PROGRAM EM03_PlacingArea_2
VAR
//----Motor-----
	// Box Placing Roller Conveyor 2	
	FB_BoxPlacingRollerConv_2			: MotorManagement;
	stBoxPlacingRollerConv_2			: stMotor;
	BoxPlacingRollerConv_2_ErrorID		: UINT;
	BoxPlacingRollerConv_2_Error		: BOOL;
	bFL_BoxPlacingRollerConv_2_Forward	: BOOL;
	bFL_BoxPlacingRollerConv_2_Reverse	: BOOL;
END_VAR

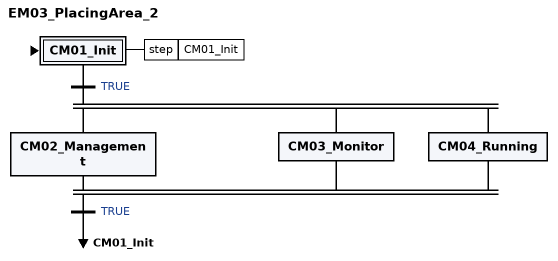
INITIAL_STEP CM01_Init:
    CM01_Init(N);  // step action
END_STEP
TRANSITION FROM CM01_Init TO (CM02_Management, CM03_Monitor, CM04_Running)
    := TRUE;
END_TRANSITION
STEP CM02_Management:
END_STEP
STEP CM03_Monitor:
END_STEP
STEP CM04_Running:
END_STEP
TRANSITION FROM (CM02_Management, CM03_Monitor, CM04_Running) TO CM01_Init
    := TRUE;
END_TRANSITION

ACTION CM01_Init:

END_ACTION

ACTION CM02_Management:
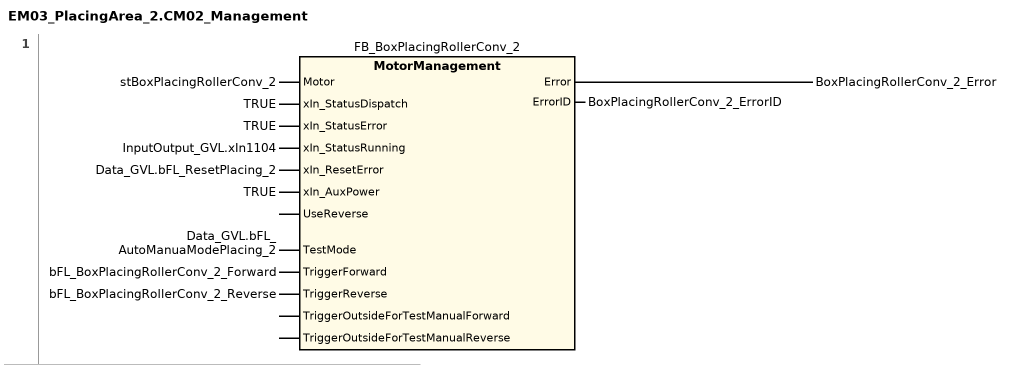
// NETWORK 1
FB_BoxPlacingRollerConv_2(
    Motor := stBoxPlacingRollerConv_2,
    xIn_StatusDispatch := TRUE,
    xIn_StatusError := TRUE,
    xIn_StatusRunning := InputOutput_GVL.xIn1104,
    xIn_ResetError := Data_GVL.bFL_ResetPlacing_2,
    xIn_AuxPower := TRUE,
    TestMode := Data_GVL.bFL_AutoManuaModePlacing_2,
    TriggerForward := bFL_BoxPlacingRollerConv_2_Forward,
    TriggerReverse := bFL_BoxPlacingRollerConv_2_Reverse,
    ErrorID => BoxPlacingRollerConv_2_ErrorID); // MotorManagement
BoxPlacingRollerConv_2_Error := FB_BoxPlacingRollerConv_2.Error;
END_ACTION

ACTION CM03_Monitor:
// NETWORK 1
END_ACTION

ACTION CM04_Running:
// NETWORK 1
END_ACTION

END_PROGRAM

(* stored: Version 1.1.0.1, ProductVersion 3.1.4024.9
   POU EM03_PlacingArea_2: Id {97f0540f-658c-4840-9ecf-0f478a222fb2}, SpecialFunc None
   Action CM01_Init: Id {007313b6-8122-49c8-9e85-a934bb5497b6}
   Action CM02_Management: Id {24479d33-40a0-48b0-9c8f-fe83d94c32f5}
   Action CM03_Monitor: Id {554e090b-6fb8-457e-8905-15ef9772bdf3}
   Action CM04_Running: Id {2c0ca033-5290-4fab-9d1a-11a228a4971b} *)
